PROGRAM MAIN
VAR
END_VAR

Process();
OperationPRG();

END_PROGRAM

(* stored: Version 1.1.0.1, ProductVersion 3.1.4024.12
   POU MAIN: Id {4ba5a4f1-694f-428e-be7a-68b479cfaaa8}, SpecialFunc None *)
